FUNCTION Convert_UDINT_TO_ULINT : Hresult
VAR_INPUT
	in : UDINT;
	out : REFERENCE TO ULINT;
END_VAR
VAR
	converted : ULINT;
END_VAR
VAR CONSTANT
	INCOMPATIBLE : HRESULT := 16#9811070E;
END_VAR

converted := UDINT_TO_ULINT(in);

IF (ULINT_TO_UDINT(converted) <> in) THEN
	Convert_UDINT_TO_ULINT := INCOMPATIBLE;
	RETURN;
END_IF

out := converted;

END_FUNCTION

(* stored: Version 1.1.0.1, ProductVersion 3.1.4024.12
   POU Convert_UDINT_TO_ULINT: Id {e53fbe71-fbde-472e-804a-f7a7174604de}, SpecialFunc None *)
